(* CoDeSys 2.3 export: DPC_TM10_para.exp *)

(* Data type in Enums *)
TYPE para_e:
(*********************************************)
(*  DON'T MAKE ANY CHANGES TO THIS ENUMS!!   *)
(*    FILE WAS AUTOMATICALLY GENERATED!!     *)
(*********************************************)
(
(* Basic *)
   EEP_number_1_1_1_e          := 790,      (* 0  (0 - 2) *)
   EEP_Input_to_Output_Mode_e  := 770,      (* Not Active  (0 - 2) *)
   EEP_test_par_new_e          := 773,      (* Not Active  (0 - 2) *)
   EEP_test_params_e           := 771,      (* Not Active  (0 - 2) *)
   EEP_test_par2_e             := 772,      (* Not Active  (0 - 2) *)

(* Test Type *)
   EEP_Trimming_type_e         := 818,      (* 53  (0 - 511) *)
   EEP_Analog_type_e           := 819,      (* 245  (53 - ) *)
   EEP_Curve_Type_e            := 820,      (* 245  (66 - 67) *)
   EEP_Function_Type_e         := 821,      (* 248  (248 - 254) *)
   EEP_Percent_Type_e          := 822,      (* 0 % (0 - 1000) *)
   EEP_Ramp_Type_e             := 823,      (* 0 % (0 - 100) *)
   EEP_Switch_Type_e           := 824,      (* 1  ( - ) *)
   EEP_List_Type_e             := 825,      (* AOC  (3 - 2) *)

(* Test Number *)
   EEP_number_1_3_1_e          := 782,      (* 0 ms (0 - 30000) *)
   EEP_number_1_3_2_e          := 783,      (* 0 ms (0 - 30000) *)
   EEP_number_1_3_3_e          := 784,      (* 0 ms (0 - 30000) *)
   EEP_number_1_3_4_e          := 785,      (* 0 ms (0 - 30000) *)
   EEP_number_1_3_5_e          := 786,      (* 0 ms (0 - 30000) *)
   EEP_number_1_3_6_e          := 787,      (* 0 ms (0 - 30000) *)
   EEP_number_1_3_7_e          := 788,      (* 0 ms (0 - 30000) *)
   EEP_number_1_3_8_e          := 789,      (* 0 ms (0 - 30000) *)

(* Output Cfg 1-8 *)
   EEP_Out_Cfg_01_e            := 832,      (* PWM  (1 - 2) *)
   EEP_Out_Cfg_02_e            := 833,      (* PWM  (1 - 2) *)
   EEP_Out_Cfg_03_e            := 834,      (* PWM  (1 - 2) *)
   EEP_Out_Cfg_04_e            := 835,      (* PWM  (1 - 2) *)
   EEP_Out_Cfg_05_e            := 836,      (* PWM  (1 - 2) *)
   EEP_Out_Cfg_06_e            := 837,      (* PWM  (1 - 2) *)
   EEP_Out_Cfg_07_e            := 838,      (* PWM  (1 - 2) *)
   EEP_Out_Cfg_08_e            := 839,      (* PWM  (1 - 2) *)

(* Output Cfg 9-16 *)
   EEP_Out_Cfg_09_e            := 840,      (* PWM  (1 - 2) *)
   EEP_Out_Cfg_10_e            := 841,      (* PWM  (1 - 2) *)
   EEP_Out_Cfg_11_e            := 842,      (* PWM  (1 - 2) *)
   EEP_Out_Cfg_12_e            := 843,      (* PWM  (1 - 2) *)
   EEP_Out_Cfg_13_e            := 844,      (* PWM  (1 - 2) *)
   EEP_Out_Cfg_14_e            := 845,      (* PWM  (1 - 2) *)
   EEP_Out_Cfg_15_e            := 846,      (* PWM  (1 - 2) *)
   EEP_Out_Cfg_16_e            := 847,      (* PWM  (1 - 2) *)

(* Output Cfg 17-24 *)
   EEP_Out_Cfg_17_e            := 848,      (* PWM  (1 - 2) *)
   EEP_Out_Cfg_18_e            := 849,      (* PWM  (1 - 2) *)
   EEP_Out_Cfg_19_e            := 850,      (* Not Active  (0 - 2) *)
   EEP_Out_Cfg_20_e            := 851,      (* Not Active  (0 - 2) *)
   EEP_Out_Cfg_21_e            := 852,      (* Not Active  (0 - 2) *)
   EEP_Out_Cfg_22_e            := 853,      (* Not Active  (0 - 2) *)
   EEP_Out_Cfg_23_e            := 854,      (* Not Active  (0 - 2) *)
   EEP_Out_Cfg_24_e            := 855,      (* Not Active  (0 - 2) *)

(* Output Cfg 25-32 *)
   EEP_Out_Cfg_25_e            := 856,      (* Not Active  (0 - 2) *)
   EEP_Out_Cfg_26_e            := 857,      (* Not Active  (0 - 2) *)
   EEP_Out_Cfg_27_e            := 858,      (* Not Active  (0 - 2) *)
   EEP_Out_Cfg_28_e            := 859,      (* Not Active  (0 - 2) *)
   EEP_Out_Cfg_29_e            := 860,      (* Not Active  (0 - 2) *)
   EEP_Out_Cfg_30_e            := 861,      (* Not Active  (0 - 2) *)
   EEP_Out_Cfg_31_e            := 862,      (* Not Active  (0 - 2) *)
   EEP_Out_Cfg_32_e            := 863,      (* Not Active  (0 - 2) *)

(* Output Cfg 33-40 *)
   EEP_Out_Cfg_33_e            := 864,      (* PWM  (2 - 2) *)
   EEP_Out_Cfg_34_e            := 865,      (* PWM  (2 - 2) *)
   EEP_Out_Cfg_35_e            := 866,      (* PWM  (2 - 2) *)
   EEP_Out_Cfg_36_e            := 867,      (* PWM  (2 - 2) *)
   EEP_Out_Cfg_37_e            := 868,      (* PWM  (1 - 2) *)
   EEP_Out_Cfg_38_e            := 869,      (* PWM  (1 - 2) *)
   EEP_Out_Cfg_39_e            := 870,      (* PWM  (1 - 2) *)
   EEP_Out_Cfg_40_e            := 871,      (* PWM  (1 - 2) *)

(* Output Cfg 41-47 *)
   EEP_Out_Cfg_41_e            := 872,      (* PWM  (1 - 2) *)
   EEP_Out_Cfg_42_e            := 873,      (* PWM  (1 - 2) *)
   EEP_Out_Cfg_43_e            := 874,      (* PWM  (1 - 2) *)
   EEP_Out_Cfg_44_e            := 875,      (* PWM  (1 - 2) *)
   EEP_Out_Cfg_45_e            := 876,      (* PWM  (1 - 2) *)
   EEP_Out_Cfg_46_e            := 877,      (* PWM  (1 - 2) *)
   EEP_Out_Cfg_47_e            := 878,      (* AOV  (3 - 2) *)

(* AOV Configuration *)
   EEP_AOV_Debounce_e          := 880,      (* 200 ms (50 - 250) *)
   EEP_AOV_Freq_e              := 881,      (* 80  (0 - 5000) *)
   EEP_AOV_Res_Min_e           := 882,      (* 0 Ohm (0 - 3000) *)
   EEP_AOV_Res_Max_e           := 883,      (* 0 Ohm (0 - 3000) *)
   EEP_AOV_Kp_e                := 884,      (* 250  (0 - 2000) *)
   EEP_AOV_Ki_e                := 885,      (* 250  (0 - 500) *)

(* AOC Configuration *)
   EEP_AOC_Debounce_e          := 888,      (* 200 ms (50 - 250) *)
   EEP_AOC_Freq_e              := 889,      (* 5000  (0 - 5000) *)
   EEP_AOC_Res_Min_e           := 890,      (* 0 Ohm (0 - 3000) *)
   EEP_AOC_Res_Max_e           := 891,      (* 0 Ohm (0 - 3000) *)
   EEP_AOC_Kp_e                := 892,      (* 250  (0 - 2000) *)
   EEP_AOC_Ki_e                := 893,      (* 250  (0 - 500) *)

(* Output Value 1-8 *)
   EEP_Out_Val_01_e            := 896,      (* 0 % / mA (0 - 10000) *)
   EEP_Out_Val_02_e            := 897,      (* 0 % / mA (0 - 10000) *)
   EEP_Out_Val_03_e            := 898,      (* 0 % / mA (0 - 10000) *)
   EEP_Out_Val_04_e            := 899,      (* 0 % / mA (0 - 10000) *)
   EEP_Out_Val_05_e            := 900,      (* 0 % / mA (0 - 10000) *)
   EEP_Out_Val_06_e            := 901,      (* 0 % / mA (0 - 10000) *)
   EEP_Out_Val_07_e            := 902,      (* 0 % / mA (0 - 10000) *)
   EEP_Out_Val_08_e            := 903,      (* 0 % / mA (0 - 10000) *)

(* Output Value 9-16 *)
   EEP_Out_Val_09_e            := 904,      (* 0 % / mA (0 - 10000) *)
   EEP_Out_Val_10_e            := 905,      (* 0 % / mA (0 - 10000) *)
   EEP_Out_Val_11_e            := 906,      (* 0 % / mA (0 - 10000) *)
   EEP_Out_Val_12_e            := 907,      (* 0 % / mA (0 - 10000) *)
   EEP_Out_Val_13_e            := 908,      (* 0 % / mA (0 - 10000) *)
   EEP_Out_Val_14_e            := 909,      (* 0 % / mA (0 - 10000) *)
   EEP_Out_Val_15_e            := 910,      (* 0 % / mA (0 - 10000) *)
   EEP_Out_Val_16_e            := 911,      (* 0 % / mA (0 - 10000) *)

(* Output Value 17-36 *)
   EEP_Out_Val_17_e            := 912,      (* 0 % / mA (0 - 10000) *)
   EEP_Out_Val_18_e            := 913,      (* 0 % / mA (0 - 10000) *)
   EEP_Out_Val_33_e            := 916,      (* 0 % / mA (0 - 10000) *)
   EEP_Out_Val_34_e            := 917,      (* 0 % / mA (0 - 10000) *)
   EEP_Out_Val_35_e            := 918,      (* 0 % / mA (0 - 10000) *)
   EEP_Out_Val_36_e            := 919,      (* 0 % / mA (0 - 10000) *)

(* Output Value 37-44 *)
   EEP_Out_Val_37_e            := 920,      (* 0 % / mA (0 - 10000) *)
   EEP_Out_Val_38_e            := 921,      (* 0 % / mA (0 - 10000) *)
   EEP_Out_Val_39_e            := 922,      (* 0 % / mA (0 - 10000) *)
   EEP_Out_Val_40_e            := 923,      (* 0 % / mA (0 - 10000) *)
   EEP_Out_Val_41_e            := 924,      (* 0 % / mA (0 - 10000) *)
   EEP_Out_Val_42_e            := 925,      (* 0 % / mA (0 - 10000) *)
   EEP_Out_Val_43_e            := 926,      (* 0 % / mA (0 - 10000) *)
   EEP_Out_Val_44_e            := 927,      (* 0 % / mA (0 - 10000) *)

(* Output Value 45-47 *)
   EEP_Out_Val_45_e            := 928,      (* 0 % / mA (0 - 10000) *)
   EEP_Out_Val_46_e            := 929,      (* 0 % / mA (0 - 10000) *)
   EEP_Out_Val_47_e            := 930,      (* 0 % / mA (0 - 20000) *)

(* POH Configuration *)
   EEP_POH_Debounce_e          := 936,      (* 100 ms (50 - 250) *)
   EEP_POH_Res_Min_e           := 938,      (* 2 Ohm (0 - 3000) *)
   EEP_POH_Res_Max_e           := 939,      (* 52 Ohm (0 - 3000) *)
   EEP_POH_Kp_e                := 940,      (* 250  (0 - 2000) *)
   EEP_POH_Ki_e                := 941,      (* 250  (0 - 500) *)

(* POL Configuration *)
   EEP_POL_Debounce_e          := 944,      (* 100 ms (50 - 250) *)
   EEP_POL_Res_Min_e           := 946,      (* 2 Ohm (0 - 3000) *)
   EEP_POL_Res_Max_e           := 947,      (* 52 Ohm (0 - 3000) *)
   EEP_POL_Kp_e                := 948,      (* 250  (0 - 2000) *)
   EEP_POL_Ki_e                := 949,      (* 250  (0 - 500) *)

(* DOH Configuration *)
   EEP_DOH_Debounce_e          := 952,      (* 200 ms (50 - 250) *)
   EEP_DOH_Res_Min_e           := 954,      (* 6 Ohm (0 - 3000) *)
   EEP_DOH_Res_Max_e           := 955       (* 44 Ohm (0 - 3000) *)

);
END_TYPE

(* Data type in Structures *)
TYPE para_ts:
(***********************************************)
(*  DON'T MAKE ANY CHANGES TO THIS STRUCTURE!! *)
(*      FILE WAS AUTOMATICALLY GENERATED!!     *)
(***********************************************)
STRUCT

(* Basic *)
   number_1_1_1_s16        : INT;           (* 0  (0 - 2) *)
   Input_to_Output_Mode_s16: INT;           (* Not Active  (0 - 2) *)
   test_par_new_s16        : INT;           (* Not Active  (0 - 2) *)
   test_params_s16         : INT;           (* Not Active  (0 - 2) *)
   test_par2_s16           : INT;           (* Not Active  (0 - 2) *)

(* Test Type *)
   Trimming_type_s16       : INT;           (* 53  (0 - 511) *)
   Analog_type_s16         : INT;           (* 245  (53 - ) *)
   Curve_Type_s16          : INT;           (* 245  (66 - 67) *)
   Function_Type_s16       : INT;           (* 248  (248 - 254) *)
   Percent_Type_s16        : INT;           (* 0 % (0 - 1000) *)
   Ramp_Type_s16           : INT;           (* 0 % (0 - 100) *)
   Switch_Type_s16         : INT;           (* 1  ( - ) *)
   List_Type_s16           : INT;           (* AOC  (3 - 2) *)

(* Test Number *)
   number_1_3_1_s16        : INT;           (* 0 ms (0 - 30000) *)
   number_1_3_2_s16        : INT;           (* 0 ms (0 - 30000) *)
   number_1_3_3_s16        : INT;           (* 0 ms (0 - 30000) *)
   number_1_3_4_s16        : INT;           (* 0 ms (0 - 30000) *)
   number_1_3_5_s16        : INT;           (* 0 ms (0 - 30000) *)
   number_1_3_6_s16        : INT;           (* 0 ms (0 - 30000) *)
   number_1_3_7_s16        : INT;           (* 0 ms (0 - 30000) *)
   number_1_3_8_s16        : INT;           (* 0 ms (0 - 30000) *)

(* Output Cfg 1-8 *)
   Out_Cfg_01_s16          : INT;           (* PWM  (1 - 2) *)
   Out_Cfg_02_s16          : INT;           (* PWM  (1 - 2) *)
   Out_Cfg_03_s16          : INT;           (* PWM  (1 - 2) *)
   Out_Cfg_04_s16          : INT;           (* PWM  (1 - 2) *)
   Out_Cfg_05_s16          : INT;           (* PWM  (1 - 2) *)
   Out_Cfg_06_s16          : INT;           (* PWM  (1 - 2) *)
   Out_Cfg_07_s16          : INT;           (* PWM  (1 - 2) *)
   Out_Cfg_08_s16          : INT;           (* PWM  (1 - 2) *)

(* Output Cfg 9-16 *)
   Out_Cfg_09_s16          : INT;           (* PWM  (1 - 2) *)
   Out_Cfg_10_s16          : INT;           (* PWM  (1 - 2) *)
   Out_Cfg_11_s16          : INT;           (* PWM  (1 - 2) *)
   Out_Cfg_12_s16          : INT;           (* PWM  (1 - 2) *)
   Out_Cfg_13_s16          : INT;           (* PWM  (1 - 2) *)
   Out_Cfg_14_s16          : INT;           (* PWM  (1 - 2) *)
   Out_Cfg_15_s16          : INT;           (* PWM  (1 - 2) *)
   Out_Cfg_16_s16          : INT;           (* PWM  (1 - 2) *)

(* Output Cfg 17-24 *)
   Out_Cfg_17_s16          : INT;           (* PWM  (1 - 2) *)
   Out_Cfg_18_s16          : INT;           (* PWM  (1 - 2) *)
   Out_Cfg_19_s16          : INT;           (* Not Active  (0 - 2) *)
   Out_Cfg_20_s16          : INT;           (* Not Active  (0 - 2) *)
   Out_Cfg_21_s16          : INT;           (* Not Active  (0 - 2) *)
   Out_Cfg_22_s16          : INT;           (* Not Active  (0 - 2) *)
   Out_Cfg_23_s16          : INT;           (* Not Active  (0 - 2) *)
   Out_Cfg_24_s16          : INT;           (* Not Active  (0 - 2) *)

(* Output Cfg 25-32 *)
   Out_Cfg_25_s16          : INT;           (* Not Active  (0 - 2) *)
   Out_Cfg_26_s16          : INT;           (* Not Active  (0 - 2) *)
   Out_Cfg_27_s16          : INT;           (* Not Active  (0 - 2) *)
   Out_Cfg_28_s16          : INT;           (* Not Active  (0 - 2) *)
   Out_Cfg_29_s16          : INT;           (* Not Active  (0 - 2) *)
   Out_Cfg_30_s16          : INT;           (* Not Active  (0 - 2) *)
   Out_Cfg_31_s16          : INT;           (* Not Active  (0 - 2) *)
   Out_Cfg_32_s16          : INT;           (* Not Active  (0 - 2) *)

(* Output Cfg 33-40 *)
   Out_Cfg_33_s16          : INT;           (* PWM  (2 - 2) *)
   Out_Cfg_34_s16          : INT;           (* PWM  (2 - 2) *)
   Out_Cfg_35_s16          : INT;           (* PWM  (2 - 2) *)
   Out_Cfg_36_s16          : INT;           (* PWM  (2 - 2) *)
   Out_Cfg_37_s16          : INT;           (* PWM  (1 - 2) *)
   Out_Cfg_38_s16          : INT;           (* PWM  (1 - 2) *)
   Out_Cfg_39_s16          : INT;           (* PWM  (1 - 2) *)
   Out_Cfg_40_s16          : INT;           (* PWM  (1 - 2) *)

(* Output Cfg 41-47 *)
   Out_Cfg_41_s16          : INT;           (* PWM  (1 - 2) *)
   Out_Cfg_42_s16          : INT;           (* PWM  (1 - 2) *)
   Out_Cfg_43_s16          : INT;           (* PWM  (1 - 2) *)
   Out_Cfg_44_s16          : INT;           (* PWM  (1 - 2) *)
   Out_Cfg_45_s16          : INT;           (* PWM  (1 - 2) *)
   Out_Cfg_46_s16          : INT;           (* PWM  (1 - 2) *)
   Out_Cfg_47_s16          : INT;           (* AOV  (3 - 2) *)

(* AOV Configuration *)
   AOV_Debounce_s16        : INT;           (* 200 ms (50 - 250) *)
   AOV_Freq_s16            : INT;           (* 80  (0 - 5000) *)
   AOV_Res_Min_s16         : INT;           (* 0 Ohm (0 - 3000) *)
   AOV_Res_Max_s16         : INT;           (* 0 Ohm (0 - 3000) *)
   AOV_Kp_s16              : INT;           (* 250  (0 - 2000) *)
   AOV_Ki_s16              : INT;           (* 250  (0 - 500) *)

(* AOC Configuration *)
   AOC_Debounce_s16        : INT;           (* 200 ms (50 - 250) *)
   AOC_Freq_s16            : INT;           (* 5000  (0 - 5000) *)
   AOC_Res_Min_s16         : INT;           (* 0 Ohm (0 - 3000) *)
   AOC_Res_Max_s16         : INT;           (* 0 Ohm (0 - 3000) *)
   AOC_Kp_s16              : INT;           (* 250  (0 - 2000) *)
   AOC_Ki_s16              : INT;           (* 250  (0 - 500) *)

(* Output Value 1-8 *)
   Out_Val_01_s16          : INT;           (* 0 % / mA (0 - 10000) *)
   Out_Val_02_s16          : INT;           (* 0 % / mA (0 - 10000) *)
   Out_Val_03_s16          : INT;           (* 0 % / mA (0 - 10000) *)
   Out_Val_04_s16          : INT;           (* 0 % / mA (0 - 10000) *)
   Out_Val_05_s16          : INT;           (* 0 % / mA (0 - 10000) *)
   Out_Val_06_s16          : INT;           (* 0 % / mA (0 - 10000) *)
   Out_Val_07_s16          : INT;           (* 0 % / mA (0 - 10000) *)
   Out_Val_08_s16          : INT;           (* 0 % / mA (0 - 10000) *)

(* Output Value 9-16 *)
   Out_Val_09_s16          : INT;           (* 0 % / mA (0 - 10000) *)
   Out_Val_10_s16          : INT;           (* 0 % / mA (0 - 10000) *)
   Out_Val_11_s16          : INT;           (* 0 % / mA (0 - 10000) *)
   Out_Val_12_s16          : INT;           (* 0 % / mA (0 - 10000) *)
   Out_Val_13_s16          : INT;           (* 0 % / mA (0 - 10000) *)
   Out_Val_14_s16          : INT;           (* 0 % / mA (0 - 10000) *)
   Out_Val_15_s16          : INT;           (* 0 % / mA (0 - 10000) *)
   Out_Val_16_s16          : INT;           (* 0 % / mA (0 - 10000) *)

(* Output Value 17-36 *)
   Out_Val_17_s16          : INT;           (* 0 % / mA (0 - 10000) *)
   Out_Val_18_s16          : INT;           (* 0 % / mA (0 - 10000) *)
   Out_Val_33_s16          : INT;           (* 0 % / mA (0 - 10000) *)
   Out_Val_34_s16          : INT;           (* 0 % / mA (0 - 10000) *)
   Out_Val_35_s16          : INT;           (* 0 % / mA (0 - 10000) *)
   Out_Val_36_s16          : INT;           (* 0 % / mA (0 - 10000) *)

(* Output Value 37-44 *)
   Out_Val_37_s16          : INT;           (* 0 % / mA (0 - 10000) *)
   Out_Val_38_s16          : INT;           (* 0 % / mA (0 - 10000) *)
   Out_Val_39_s16          : INT;           (* 0 % / mA (0 - 10000) *)
   Out_Val_40_s16          : INT;           (* 0 % / mA (0 - 10000) *)
   Out_Val_41_s16          : INT;           (* 0 % / mA (0 - 10000) *)
   Out_Val_42_s16          : INT;           (* 0 % / mA (0 - 10000) *)
   Out_Val_43_s16          : INT;           (* 0 % / mA (0 - 10000) *)
   Out_Val_44_s16          : INT;           (* 0 % / mA (0 - 10000) *)

(* Output Value 45-47 *)
   Out_Val_45_s16          : INT;           (* 0 % / mA (0 - 10000) *)
   Out_Val_46_s16          : INT;           (* 0 % / mA (0 - 10000) *)
   Out_Val_47_s16          : INT;           (* 0 % / mA (0 - 20000) *)

(* POH Configuration *)
   POH_Debounce_s16        : INT;           (* 100 ms (50 - 250) *)
   POH_Res_Min_s16         : INT;           (* 2 Ohm (0 - 3000) *)
   POH_Res_Max_s16         : INT;           (* 52 Ohm (0 - 3000) *)
   POH_Kp_s16              : INT;           (* 250  (0 - 2000) *)
   POH_Ki_s16              : INT;           (* 250  (0 - 500) *)

(* POL Configuration *)
   POL_Debounce_s16        : INT;           (* 100 ms (50 - 250) *)
   POL_Res_Min_s16         : INT;           (* 2 Ohm (0 - 3000) *)
   POL_Res_Max_s16         : INT;           (* 52 Ohm (0 - 3000) *)
   POL_Kp_s16              : INT;           (* 250  (0 - 2000) *)
   POL_Ki_s16              : INT;           (* 250  (0 - 500) *)

(* DOH Configuration *)
   DOH_Debounce_s16        : INT;           (* 200 ms (50 - 250) *)
   DOH_Res_Min_s16         : INT;           (* 6 Ohm (0 - 3000) *)
   DOH_Res_Max_s16         : INT;           (* 44 Ohm (0 - 3000) *)
END_STRUCT
END_TYPE

(* POU Autocode/Callback_diag_getPara, ST *)
PROGRAM Callback_diag_getPara
VAR
   eep:  ARRAY [0..1280] OF INT;
END_VAR
(*********************************************)
(*  DON'T MAKE ANY CHANGES TO THIS PROGRAM!! *)
(*     FILE WAS AUTOMATICALLY GENERATED!!    *)
(*********************************************)

(* get EEPROM pages 0..4 *)
ree_getArray( PAGE0, 0, ADR(eep[0]),    256 );
ree_getArray( PAGE1, 0, ADR(eep[256]),  256 );
ree_getArray( PAGE2, 0, ADR(eep[512]),  256 );
ree_getArray( PAGE3, 0, ADR(eep[768]),  256 );
ree_getArray( PAGE4, 0, ADR(eep[1024]), 256 );

(* Basic *)
para_s.number_1_1_1_s16         := eep[EEP_number_1_1_1_e];
para_s.Input_to_Output_Mode_s16 := eep[EEP_Input_to_Output_Mode_e];
para_s.test_par_new_s16         := eep[EEP_test_par_new_e];
para_s.test_params_s16          := eep[EEP_test_params_e];
para_s.test_par2_s16            := eep[EEP_test_par2_e];

(* Test Type *)
para_s.Trimming_type_s16        := eep[EEP_Trimming_type_e];
para_s.Analog_type_s16          := eep[EEP_Analog_type_e];
para_s.Curve_Type_s16           := eep[EEP_Curve_Type_e];
para_s.Function_Type_s16        := eep[EEP_Function_Type_e];
para_s.Percent_Type_s16         := eep[EEP_Percent_Type_e];
para_s.Ramp_Type_s16            := eep[EEP_Ramp_Type_e];
para_s.Switch_Type_s16          := eep[EEP_Switch_Type_e];
para_s.List_Type_s16            := eep[EEP_List_Type_e];

(* Test Number *)
para_s.number_1_3_1_s16         := eep[EEP_number_1_3_1_e];
para_s.number_1_3_2_s16         := eep[EEP_number_1_3_2_e];
para_s.number_1_3_3_s16         := eep[EEP_number_1_3_3_e];
para_s.number_1_3_4_s16         := eep[EEP_number_1_3_4_e];
para_s.number_1_3_5_s16         := eep[EEP_number_1_3_5_e];
para_s.number_1_3_6_s16         := eep[EEP_number_1_3_6_e];
para_s.number_1_3_7_s16         := eep[EEP_number_1_3_7_e];
para_s.number_1_3_8_s16         := eep[EEP_number_1_3_8_e];

(* Output Cfg 1-8 *)
para_s.Out_Cfg_01_s16           := eep[EEP_Out_Cfg_01_e];
para_s.Out_Cfg_02_s16           := eep[EEP_Out_Cfg_02_e];
para_s.Out_Cfg_03_s16           := eep[EEP_Out_Cfg_03_e];
para_s.Out_Cfg_04_s16           := eep[EEP_Out_Cfg_04_e];
para_s.Out_Cfg_05_s16           := eep[EEP_Out_Cfg_05_e];
para_s.Out_Cfg_06_s16           := eep[EEP_Out_Cfg_06_e];
para_s.Out_Cfg_07_s16           := eep[EEP_Out_Cfg_07_e];
para_s.Out_Cfg_08_s16           := eep[EEP_Out_Cfg_08_e];

(* Output Cfg 9-16 *)
para_s.Out_Cfg_09_s16           := eep[EEP_Out_Cfg_09_e];
para_s.Out_Cfg_10_s16           := eep[EEP_Out_Cfg_10_e];
para_s.Out_Cfg_11_s16           := eep[EEP_Out_Cfg_11_e];
para_s.Out_Cfg_12_s16           := eep[EEP_Out_Cfg_12_e];
para_s.Out_Cfg_13_s16           := eep[EEP_Out_Cfg_13_e];
para_s.Out_Cfg_14_s16           := eep[EEP_Out_Cfg_14_e];
para_s.Out_Cfg_15_s16           := eep[EEP_Out_Cfg_15_e];
para_s.Out_Cfg_16_s16           := eep[EEP_Out_Cfg_16_e];

(* Output Cfg 17-24 *)
para_s.Out_Cfg_17_s16           := eep[EEP_Out_Cfg_17_e];
para_s.Out_Cfg_18_s16           := eep[EEP_Out_Cfg_18_e];
para_s.Out_Cfg_19_s16           := eep[EEP_Out_Cfg_19_e];
para_s.Out_Cfg_20_s16           := eep[EEP_Out_Cfg_20_e];
para_s.Out_Cfg_21_s16           := eep[EEP_Out_Cfg_21_e];
para_s.Out_Cfg_22_s16           := eep[EEP_Out_Cfg_22_e];
para_s.Out_Cfg_23_s16           := eep[EEP_Out_Cfg_23_e];
para_s.Out_Cfg_24_s16           := eep[EEP_Out_Cfg_24_e];

(* Output Cfg 25-32 *)
para_s.Out_Cfg_25_s16           := eep[EEP_Out_Cfg_25_e];
para_s.Out_Cfg_26_s16           := eep[EEP_Out_Cfg_26_e];
para_s.Out_Cfg_27_s16           := eep[EEP_Out_Cfg_27_e];
para_s.Out_Cfg_28_s16           := eep[EEP_Out_Cfg_28_e];
para_s.Out_Cfg_29_s16           := eep[EEP_Out_Cfg_29_e];
para_s.Out_Cfg_30_s16           := eep[EEP_Out_Cfg_30_e];
para_s.Out_Cfg_31_s16           := eep[EEP_Out_Cfg_31_e];
para_s.Out_Cfg_32_s16           := eep[EEP_Out_Cfg_32_e];

(* Output Cfg 33-40 *)
para_s.Out_Cfg_33_s16           := eep[EEP_Out_Cfg_33_e];
para_s.Out_Cfg_34_s16           := eep[EEP_Out_Cfg_34_e];
para_s.Out_Cfg_35_s16           := eep[EEP_Out_Cfg_35_e];
para_s.Out_Cfg_36_s16           := eep[EEP_Out_Cfg_36_e];
para_s.Out_Cfg_37_s16           := eep[EEP_Out_Cfg_37_e];
para_s.Out_Cfg_38_s16           := eep[EEP_Out_Cfg_38_e];
para_s.Out_Cfg_39_s16           := eep[EEP_Out_Cfg_39_e];
para_s.Out_Cfg_40_s16           := eep[EEP_Out_Cfg_40_e];

(* Output Cfg 41-47 *)
para_s.Out_Cfg_41_s16           := eep[EEP_Out_Cfg_41_e];
para_s.Out_Cfg_42_s16           := eep[EEP_Out_Cfg_42_e];
para_s.Out_Cfg_43_s16           := eep[EEP_Out_Cfg_43_e];
para_s.Out_Cfg_44_s16           := eep[EEP_Out_Cfg_44_e];
para_s.Out_Cfg_45_s16           := eep[EEP_Out_Cfg_45_e];
para_s.Out_Cfg_46_s16           := eep[EEP_Out_Cfg_46_e];
para_s.Out_Cfg_47_s16           := eep[EEP_Out_Cfg_47_e];

(* AOV Configuration *)
para_s.AOV_Debounce_s16         := eep[EEP_AOV_Debounce_e];
para_s.AOV_Freq_s16             := eep[EEP_AOV_Freq_e];
para_s.AOV_Res_Min_s16          := eep[EEP_AOV_Res_Min_e];
para_s.AOV_Res_Max_s16          := eep[EEP_AOV_Res_Max_e];
para_s.AOV_Kp_s16               := eep[EEP_AOV_Kp_e];
para_s.AOV_Ki_s16               := eep[EEP_AOV_Ki_e];

(* AOC Configuration *)
para_s.AOC_Debounce_s16         := eep[EEP_AOC_Debounce_e];
para_s.AOC_Freq_s16             := eep[EEP_AOC_Freq_e];
para_s.AOC_Res_Min_s16          := eep[EEP_AOC_Res_Min_e];
para_s.AOC_Res_Max_s16          := eep[EEP_AOC_Res_Max_e];
para_s.AOC_Kp_s16               := eep[EEP_AOC_Kp_e];
para_s.AOC_Ki_s16               := eep[EEP_AOC_Ki_e];

(* Output Value 1-8 *)
para_s.Out_Val_01_s16           := eep[EEP_Out_Val_01_e];
para_s.Out_Val_02_s16           := eep[EEP_Out_Val_02_e];
para_s.Out_Val_03_s16           := eep[EEP_Out_Val_03_e];
para_s.Out_Val_04_s16           := eep[EEP_Out_Val_04_e];
para_s.Out_Val_05_s16           := eep[EEP_Out_Val_05_e];
para_s.Out_Val_06_s16           := eep[EEP_Out_Val_06_e];
para_s.Out_Val_07_s16           := eep[EEP_Out_Val_07_e];
para_s.Out_Val_08_s16           := eep[EEP_Out_Val_08_e];

(* Output Value 9-16 *)
para_s.Out_Val_09_s16           := eep[EEP_Out_Val_09_e];
para_s.Out_Val_10_s16           := eep[EEP_Out_Val_10_e];
para_s.Out_Val_11_s16           := eep[EEP_Out_Val_11_e];
para_s.Out_Val_12_s16           := eep[EEP_Out_Val_12_e];
para_s.Out_Val_13_s16           := eep[EEP_Out_Val_13_e];
para_s.Out_Val_14_s16           := eep[EEP_Out_Val_14_e];
para_s.Out_Val_15_s16           := eep[EEP_Out_Val_15_e];
para_s.Out_Val_16_s16           := eep[EEP_Out_Val_16_e];

(* Output Value 17-36 *)
para_s.Out_Val_17_s16           := eep[EEP_Out_Val_17_e];
para_s.Out_Val_18_s16           := eep[EEP_Out_Val_18_e];
para_s.Out_Val_33_s16           := eep[EEP_Out_Val_33_e];
para_s.Out_Val_34_s16           := eep[EEP_Out_Val_34_e];
para_s.Out_Val_35_s16           := eep[EEP_Out_Val_35_e];
para_s.Out_Val_36_s16           := eep[EEP_Out_Val_36_e];

(* Output Value 37-44 *)
para_s.Out_Val_37_s16           := eep[EEP_Out_Val_37_e];
para_s.Out_Val_38_s16           := eep[EEP_Out_Val_38_e];
para_s.Out_Val_39_s16           := eep[EEP_Out_Val_39_e];
para_s.Out_Val_40_s16           := eep[EEP_Out_Val_40_e];
para_s.Out_Val_41_s16           := eep[EEP_Out_Val_41_e];
para_s.Out_Val_42_s16           := eep[EEP_Out_Val_42_e];
para_s.Out_Val_43_s16           := eep[EEP_Out_Val_43_e];
para_s.Out_Val_44_s16           := eep[EEP_Out_Val_44_e];

(* Output Value 45-47 *)
para_s.Out_Val_45_s16           := eep[EEP_Out_Val_45_e];
para_s.Out_Val_46_s16           := eep[EEP_Out_Val_46_e];
para_s.Out_Val_47_s16           := eep[EEP_Out_Val_47_e];

(* POH Configuration *)
para_s.POH_Debounce_s16         := eep[EEP_POH_Debounce_e];
para_s.POH_Res_Min_s16          := eep[EEP_POH_Res_Min_e];
para_s.POH_Res_Max_s16          := eep[EEP_POH_Res_Max_e];
para_s.POH_Kp_s16               := eep[EEP_POH_Kp_e];
para_s.POH_Ki_s16               := eep[EEP_POH_Ki_e];

(* POL Configuration *)
para_s.POL_Debounce_s16         := eep[EEP_POL_Debounce_e];
para_s.POL_Res_Min_s16          := eep[EEP_POL_Res_Min_e];
para_s.POL_Res_Max_s16          := eep[EEP_POL_Res_Max_e];
para_s.POL_Kp_s16               := eep[EEP_POL_Kp_e];
para_s.POL_Ki_s16               := eep[EEP_POL_Ki_e];

(* DOH Configuration *)
para_s.DOH_Debounce_s16         := eep[EEP_DOH_Debounce_e];
para_s.DOH_Res_Min_s16          := eep[EEP_DOH_Res_Min_e];
para_s.DOH_Res_Max_s16          := eep[EEP_DOH_Res_Max_e];
END_PROGRAM

(* POU Autocode/PrmData, ST *)
PROGRAM PrmData
(*********************************************)
(*  DON'T MAKE ANY CHANGES TO THIS PROGRAM!! *)
(*     FILE WAS AUTOMATICALLY GENERATED!!    *)
(*********************************************)

VAR
END_VAR
VAR CONSTANT

(**)
(*********************************************)
nrPrmMenus_u8          : USINT := 5;

(*********************************************)
(* Parameters Tree *)
(*********************************************)

ParameterMenus_as      : ARRAY [1..5] OF ParameterMenu_ts := 

   (*********************************************)
   (* parameter menu 1 - up to 8 groups can be defined here *)
   (*********************************************)
   (
      MenuName_as8        := 'Menu 1',

      ParameterGroup_as   := 

      (*********************************************)
      (* parameter group 1.1 - up to 8 parameters can be defined here *)
      (*********************************************)
      (
         GroupName_as8   := 'Basic',

         Param_as        := 

         (*********************************************)
         (* parameter 1.1.1 *)
         (*********************************************)
         (
            ParameterName_as8    := 'List test 1',
            ParameterType_u8     := 0,
            attr1_u              := 0,
            attr2_u              := 2,
            UnitCode_au8         := 0,
            AccesslevelCode_u8   := 129,
            attr4_u              := 0,
            EEPROMAddress_s      := (Page_u8 := 3, IntIndex_u8 := 22)
         ),

         (*********************************************)
         (* parameter 1.1.2 *)
         (*********************************************)
         (
            ParameterName_as8    := 'Input_to_Output_Mode',
            ParameterType_u8     := 7,
            attr1_u              := 0,
            attr2_u              := 2,
            UnitCode_au8         := 0,
            AccesslevelCode_u8   := 129,
            attr4_u              := 0,
            EEPROMAddress_s      := (Page_u8 := 3, IntIndex_u8 := 2)
         ),

         (*********************************************)
         (* parameter 1.1.3 *)
         (*********************************************)
         (
         ),

         (*********************************************)
         (* parameter 1.1.4 *)
         (*********************************************)
         (
            ParameterName_as8    := 'Test parameter new',
            ParameterType_u8     := 7,
            attr1_u              := 0,
            attr2_u              := 2,
            UnitCode_au8         := 0,
            AccesslevelCode_u8   := 129,
            attr4_u              := 0,
            EEPROMAddress_s      := (Page_u8 := 3, IntIndex_u8 := 5)
         ),

         (*********************************************)
         (* parameter 1.1.5 *)
         (*********************************************)
         (
         ),

         (*********************************************)
         (* parameter 1.1.6 *)
         (*********************************************)
         (
            ParameterName_as8    := 'Test_parameter',
            ParameterType_u8     := 7,
            attr1_u              := 0,
            attr2_u              := 2,
            UnitCode_au8         := 0,
            AccesslevelCode_u8   := 129,
            attr4_u              := 0,
            EEPROMAddress_s      := (Page_u8 := 3, IntIndex_u8 := 3)
         ),

         (*********************************************)
         (* parameter 1.1.7 *)
         (*********************************************)
         (
         ),

         (*********************************************)
         (* parameter 1.1.8 *)
         (*********************************************)
         (
            ParameterName_as8    := 'Test_params',
            ParameterType_u8     := 7,
            attr1_u              := 0,
            attr2_u              := 2,
            UnitCode_au8         := 0,
            AccesslevelCode_u8   := 129,
            attr4_u              := 0,
            EEPROMAddress_s      := (Page_u8 := 3, IntIndex_u8 := 4)
         )

      ),

      (*********************************************)
      (* parameter group 1.2 - up to 8 parameters can be defined here *)
      (*********************************************)
      (
         GroupName_as8   := 'Test Type',

         Param_as        := 

         (*********************************************)
         (* parameter 1.2.1 *)
         (*********************************************)
         (
            ParameterName_as8    := 'Trimming type',
            ParameterType_u8     := 5,
            attr1_u              := 0,
            attr2_u              := 511,
            UnitCode_au8         := 0,
            AccesslevelCode_u8   := 129,
            attr4_u              := 0,
            EEPROMAddress_s      := (Page_u8 := 3, IntIndex_u8 := 50)
         ),

         (*********************************************)
         (* parameter 1.2.2 *)
         (*********************************************)
         (
            ParameterName_as8    := 'Analog type',
            ParameterType_u8     := 8,
            attr1_u              := 53,
            UnitCode_au8         := 0,
            AccesslevelCode_u8   := 129,
            attr4_u              := 249,
            EEPROMAddress_s      := (Page_u8 := 3, IntIndex_u8 := 51)
         ),

         (*********************************************)
         (* parameter 1.2.3 *)
         (*********************************************)
         (
            ParameterName_as8    := 'Curve Type',
            ParameterType_u8     := 6,
            attr1_u              := 66,
            attr2_u              := 67,
            attr3_u              := 3000,
            UnitCode_au8         := 0,
            AccesslevelCode_u8   := 129,
            attr4_u              := 245,
            EEPROMAddress_s      := (Page_u8 := 3, IntIndex_u8 := 52)
         ),

         (*********************************************)
         (* parameter 1.2.4 *)
         (*********************************************)
         (
            ParameterName_as8    := 'Function Type',
            ParameterType_u8     := 9,
            attr1_u              := 248,
            attr2_u              := 254,
            attr3_u              := 248,
            UnitCode_au8         := 0,
            AccesslevelCode_u8   := 129,
            attr4_u              := 248,
            EEPROMAddress_s      := (Page_u8 := 3, IntIndex_u8 := 53)
         ),

         (*********************************************)
         (* parameter 1.2.5 *)
         (*********************************************)
         (
            ParameterName_as8    := 'Percent Type',
            ParameterType_u8     := 0,
            attr1_u              := 0,
            attr2_u              := 1000,
            attr3_u              := 10,
            UnitCode_au8         := 1,
            Multiplier_s16       := 1,
            Divisor_s16          := 1,
            NumberOfDigits_u16   := 0,
            AccesslevelCode_u8   := 129,
            attr4_u              := 0,
            EEPROMAddress_s      := (Page_u8 := 3, IntIndex_u8 := 54)
         ),

         (*********************************************)
         (* parameter 1.2.6 *)
         (*********************************************)
         (
            ParameterName_as8    := 'Ramp Type',
            ParameterType_u8     := 0,
            attr1_u              := 0,
            attr2_u              := 100,
            attr3_u              := 10,
            UnitCode_au8         := 1,
            Multiplier_s16       := 1,
            Divisor_s16          := 1,
            NumberOfDigits_u16   := 0,
            AccesslevelCode_u8   := 129,
            attr4_u              := 0,
            EEPROMAddress_s      := (Page_u8 := 3, IntIndex_u8 := 55)
         ),

         (*********************************************)
         (* parameter 1.2.7 *)
         (*********************************************)
         (
            ParameterName_as8    := 'Switch Type',
            ParameterType_u8     := 4,
            UnitCode_au8         := 0,
            AccesslevelCode_u8   := 129,
            attr4_u              := 1,
            EEPROMAddress_s      := (Page_u8 := 3, IntIndex_u8 := 56)
         ),

         (*********************************************)
         (* parameter 1.2.8 *)
         (*********************************************)
         (
            ParameterName_as8    := 'List Type',
            ParameterType_u8     := 7,
            attr1_u              := 3,
            attr2_u              := 2,
            UnitCode_au8         := 0,
            AccesslevelCode_u8   := 129,
            attr4_u              := 0,
            EEPROMAddress_s      := (Page_u8 := 3, IntIndex_u8 := 57)
         )

      ),

      (*********************************************)
      (* parameter group 1.3 - up to 8 parameters can be defined here *)
      (*********************************************)
      (
         GroupName_as8   := 'Test Number',

         Param_as        := 

         (*********************************************)
         (* parameter 1.3.1 *)
         (*********************************************)
         (
            ParameterName_as8    := 'Number test 1',
            ParameterType_u8     := 0,
            attr1_u              := 0,
            attr2_u              := 30000,
            attr3_u              := 1,
            UnitCode_au8         := 4,
            Multiplier_s16       := 1,
            Divisor_s16          := 1,
            NumberOfDigits_u16   := 0,
            AccesslevelCode_u8   := 129,
            attr4_u              := 0,
            EEPROMAddress_s      := (Page_u8 := 3, IntIndex_u8 := 14)
         ),

         (*********************************************)
         (* parameter 1.3.2 *)
         (*********************************************)
         (
            ParameterName_as8    := 'Number test 2',
            ParameterType_u8     := 0,
            attr1_u              := 0,
            attr2_u              := 30000,
            attr3_u              := 1,
            UnitCode_au8         := 4,
            Multiplier_s16       := 1,
            Divisor_s16          := 1,
            NumberOfDigits_u16   := 0,
            AccesslevelCode_u8   := 129,
            attr4_u              := 0,
            EEPROMAddress_s      := (Page_u8 := 3, IntIndex_u8 := 15)
         ),

         (*********************************************)
         (* parameter 1.3.3 *)
         (*********************************************)
         (
            ParameterName_as8    := 'Number test 3',
            ParameterType_u8     := 0,
            attr1_u              := 0,
            attr2_u              := 30000,
            attr3_u              := 1,
            UnitCode_au8         := 4,
            Multiplier_s16       := 1,
            Divisor_s16          := 1,
            NumberOfDigits_u16   := 0,
            AccesslevelCode_u8   := 129,
            attr4_u              := 0,
            EEPROMAddress_s      := (Page_u8 := 3, IntIndex_u8 := 16)
         ),

         (*********************************************)
         (* parameter 1.3.4 *)
         (*********************************************)
         (
            ParameterName_as8    := 'Number test 4',
            ParameterType_u8     := 0,
            attr1_u              := 0,
            attr2_u              := 30000,
            attr3_u              := 1,
            UnitCode_au8         := 4,
            Multiplier_s16       := 1,
            Divisor_s16          := 1,
            NumberOfDigits_u16   := 0,
            AccesslevelCode_u8   := 129,
            attr4_u              := 0,
            EEPROMAddress_s      := (Page_u8 := 3, IntIndex_u8 := 17)
         ),

         (*********************************************)
         (* parameter 1.3.5 *)
         (*********************************************)
         (
            ParameterName_as8    := 'Number test 5',
            ParameterType_u8     := 0,
            attr1_u              := 0,
            attr2_u              := 30000,
            attr3_u              := 1,
            UnitCode_au8         := 4,
            Multiplier_s16       := 1,
            Divisor_s16          := 1,
            NumberOfDigits_u16   := 0,
            AccesslevelCode_u8   := 129,
            attr4_u              := 0,
            EEPROMAddress_s      := (Page_u8 := 3, IntIndex_u8 := 18)
         ),

         (*********************************************)
         (* parameter 1.3.6 *)
         (*********************************************)
         (
            ParameterName_as8    := 'Number test 6',
            ParameterType_u8     := 0,
            attr1_u              := 0,
            attr2_u              := 30000,
            attr3_u              := 1,
            UnitCode_au8         := 4,
            Multiplier_s16       := 1,
            Divisor_s16          := 1,
            NumberOfDigits_u16   := 0,
            AccesslevelCode_u8   := 129,
            attr4_u              := 0,
            EEPROMAddress_s      := (Page_u8 := 3, IntIndex_u8 := 19)
         ),

         (*********************************************)
         (* parameter 1.3.7 *)
         (*********************************************)
         (
            ParameterName_as8    := 'Number test 7',
            ParameterType_u8     := 0,
            attr1_u              := 0,
            attr2_u              := 30000,
            attr3_u              := 1,
            UnitCode_au8         := 4,
            Multiplier_s16       := 1,
            Divisor_s16          := 1,
            NumberOfDigits_u16   := 0,
            AccesslevelCode_u8   := 129,
            attr4_u              := 0,
            EEPROMAddress_s      := (Page_u8 := 3, IntIndex_u8 := 20)
         ),

         (*********************************************)
         (* parameter 1.3.8 *)
         (*********************************************)
         (
            ParameterName_as8    := 'Number test 8',
            ParameterType_u8     := 0,
            attr1_u              := 0,
            attr2_u              := 30000,
            attr3_u              := 1,
            UnitCode_au8         := 4,
            Multiplier_s16       := 1,
            Divisor_s16          := 1,
            NumberOfDigits_u16   := 0,
            AccesslevelCode_u8   := 129,
            attr4_u              := 0,
            EEPROMAddress_s      := (Page_u8 := 3, IntIndex_u8 := 21)
         )

      ),

      (*********************************************)
      (* parameter group 1.4 - up to 8 parameters can be defined here *)
      (*********************************************)
      (








      ),

      (*********************************************)
      (* parameter group 1.5 - up to 8 parameters can be defined here *)
      (*********************************************)
      (








      ),

      (*********************************************)
      (* parameter group 1.6 - up to 8 parameters can be defined here *)
      (*********************************************)
      (








      ),

      (*********************************************)
      (* parameter group 1.7 - up to 8 parameters can be defined here *)
      (*********************************************)
      (








      ),

      (*********************************************)
      (* parameter group 1.8 - up to 8 parameters can be defined here *)
      (*********************************************)
      (








      )

   ),

   (*********************************************)
   (* parameter menu 2 - up to 8 groups can be defined here *)
   (*********************************************)
   (
      MenuName_as8        := 'Menu 2',

      ParameterGroup_as   := 

      (*********************************************)
      (* parameter group 2.1 - up to 8 parameters can be defined here *)
      (*********************************************)
      (
         GroupName_as8   := 'Output Cfg 1-8',

         Param_as        := 

         (*********************************************)
         (* parameter 2.1.1 *)
         (*********************************************)
         (
            ParameterName_as8    := 'Output Cfg 1',
            ParameterType_u8     := 7,
            attr1_u              := 1,
            attr2_u              := 2,
            UnitCode_au8         := 0,
            AccesslevelCode_u8   := 129,
            attr4_u              := 0,
            EEPROMAddress_s      := (Page_u8 := 3, IntIndex_u8 := 64)
         ),

         (*********************************************)
         (* parameter 2.1.2 *)
         (*********************************************)
         (
            ParameterName_as8    := 'Output Cfg 2',
            ParameterType_u8     := 7,
            attr1_u              := 1,
            attr2_u              := 2,
            UnitCode_au8         := 0,
            AccesslevelCode_u8   := 129,
            attr4_u              := 0,
            EEPROMAddress_s      := (Page_u8 := 3, IntIndex_u8 := 65)
         ),

         (*********************************************)
         (* parameter 2.1.3 *)
         (*********************************************)
         (
            ParameterName_as8    := 'Output Cfg 3',
            ParameterType_u8     := 7,
            attr1_u              := 1,
            attr2_u              := 2,
            UnitCode_au8         := 0,
            AccesslevelCode_u8   := 129,
            attr4_u              := 0,
            EEPROMAddress_s      := (Page_u8 := 3, IntIndex_u8 := 66)
         ),

         (*********************************************)
         (* parameter 2.1.4 *)
         (*********************************************)
         (
            ParameterName_as8    := 'Output Cfg 4',
            ParameterType_u8     := 7,
            attr1_u              := 1,
            attr2_u              := 2,
            UnitCode_au8         := 0,
            AccesslevelCode_u8   := 129,
            attr4_u              := 0,
            EEPROMAddress_s      := (Page_u8 := 3, IntIndex_u8 := 67)
         ),

         (*********************************************)
         (* parameter 2.1.5 *)
         (*********************************************)
         (
            ParameterName_as8    := 'Output Cfg 5',
            ParameterType_u8     := 7,
            attr1_u              := 1,
            attr2_u              := 2,
            UnitCode_au8         := 0,
            AccesslevelCode_u8   := 129,
            attr4_u              := 0,
            EEPROMAddress_s      := (Page_u8 := 3, IntIndex_u8 := 68)
         ),

         (*********************************************)
         (* parameter 2.1.6 *)
         (*********************************************)
         (
            ParameterName_as8    := 'Output Cfg 6',
            ParameterType_u8     := 7,
            attr1_u              := 1,
            attr2_u              := 2,
            UnitCode_au8         := 0,
            AccesslevelCode_u8   := 129,
            attr4_u              := 0,
            EEPROMAddress_s      := (Page_u8 := 3, IntIndex_u8 := 69)
         ),

         (*********************************************)
         (* parameter 2.1.7 *)
         (*********************************************)
         (
            ParameterName_as8    := 'Output Cfg 7',
            ParameterType_u8     := 7,
            attr1_u              := 1,
            attr2_u              := 2,
            UnitCode_au8         := 0,
            AccesslevelCode_u8   := 129,
            attr4_u              := 0,
            EEPROMAddress_s      := (Page_u8 := 3, IntIndex_u8 := 70)
         ),

         (*********************************************)
         (* parameter 2.1.8 *)
         (*********************************************)
         (
            ParameterName_as8    := 'Output Cfg 8',
            ParameterType_u8     := 7,
            attr1_u              := 1,
            attr2_u              := 2,
            UnitCode_au8         := 0,
            AccesslevelCode_u8   := 129,
            attr4_u              := 0,
            EEPROMAddress_s      := (Page_u8 := 3, IntIndex_u8 := 71)
         )

      ),

      (*********************************************)
      (* parameter group 2.2 - up to 8 parameters can be defined here *)
      (*********************************************)
      (
         GroupName_as8   := 'Output Cfg 9-16',

         Param_as        := 

         (*********************************************)
         (* parameter 2.2.1 *)
         (*********************************************)
         (
            ParameterName_as8    := 'Output Cfg 9',
            ParameterType_u8     := 7,
            attr1_u              := 1,
            attr2_u              := 2,
            UnitCode_au8         := 0,
            AccesslevelCode_u8   := 129,
            attr4_u              := 0,
            EEPROMAddress_s      := (Page_u8 := 3, IntIndex_u8 := 72)
         ),

         (*********************************************)
         (* parameter 2.2.2 *)
         (*********************************************)
         (
            ParameterName_as8    := 'Output Cfg 10',
            ParameterType_u8     := 7,
            attr1_u              := 1,
            attr2_u              := 2,
            UnitCode_au8         := 0,
            AccesslevelCode_u8   := 129,
            attr4_u              := 0,
            EEPROMAddress_s      := (Page_u8 := 3, IntIndex_u8 := 73)
         ),

         (*********************************************)
         (* parameter 2.2.3 *)
         (*********************************************)
         (
            ParameterName_as8    := 'Output Cfg 11',
            ParameterType_u8     := 7,
            attr1_u              := 1,
            attr2_u              := 2,
            UnitCode_au8         := 0,
            AccesslevelCode_u8   := 129,
            attr4_u              := 0,
            EEPROMAddress_s      := (Page_u8 := 3, IntIndex_u8 := 74)
         ),

         (*********************************************)
         (* parameter 2.2.4 *)
         (*********************************************)
         (
            ParameterName_as8    := 'Output Cfg 12',
            ParameterType_u8     := 7,
            attr1_u              := 1,
            attr2_u              := 2,
            UnitCode_au8         := 0,
            AccesslevelCode_u8   := 129,
            attr4_u              := 0,
            EEPROMAddress_s      := (Page_u8 := 3, IntIndex_u8 := 75)
         ),

         (*********************************************)
         (* parameter 2.2.5 *)
         (*********************************************)
         (
            ParameterName_as8    := 'Output Cfg 13',
            ParameterType_u8     := 7,
            attr1_u              := 1,
            attr2_u              := 2,
            UnitCode_au8         := 0,
            AccesslevelCode_u8   := 129,
            attr4_u              := 0,
            EEPROMAddress_s      := (Page_u8 := 3, IntIndex_u8 := 76)
         ),

         (*********************************************)
         (* parameter 2.2.6 *)
         (*********************************************)
         (
            ParameterName_as8    := 'Output Cfg 14',
            ParameterType_u8     := 7,
            attr1_u              := 1,
            attr2_u              := 2,
            UnitCode_au8         := 0,
            AccesslevelCode_u8   := 129,
            attr4_u              := 0,
            EEPROMAddress_s      := (Page_u8 := 3, IntIndex_u8 := 77)
         ),

         (*********************************************)
         (* parameter 2.2.7 *)
         (*********************************************)
         (
            ParameterName_as8    := 'Output Cfg 15',
            ParameterType_u8     := 7,
            attr1_u              := 1,
            attr2_u              := 2,
            UnitCode_au8         := 0,
            AccesslevelCode_u8   := 129,
            attr4_u              := 0,
            EEPROMAddress_s      := (Page_u8 := 3, IntIndex_u8 := 78)
         ),

         (*********************************************)
         (* parameter 2.2.8 *)
         (*********************************************)
         (
            ParameterName_as8    := 'Output Cfg 16',
            ParameterType_u8     := 7,
            attr1_u              := 1,
            attr2_u              := 2,
            UnitCode_au8         := 0,
            AccesslevelCode_u8   := 129,
            attr4_u              := 0,
            EEPROMAddress_s      := (Page_u8 := 3, IntIndex_u8 := 79)
         )

      ),

      (*********************************************)
      (* parameter group 2.3 - up to 8 parameters can be defined here *)
      (*********************************************)
      (
         GroupName_as8   := 'Output Cfg 17-24',

         Param_as        := 

         (*********************************************)
         (* parameter 2.3.1 *)
         (*********************************************)
         (
            ParameterName_as8    := 'Output Cfg 17',
            ParameterType_u8     := 7,
            attr1_u              := 1,
            attr2_u              := 2,
            UnitCode_au8         := 0,
            AccesslevelCode_u8   := 129,
            attr4_u              := 0,
            EEPROMAddress_s      := (Page_u8 := 3, IntIndex_u8 := 80)
         ),

         (*********************************************)
         (* parameter 2.3.2 *)
         (*********************************************)
         (
            ParameterName_as8    := 'Output Cfg 18',
            ParameterType_u8     := 7,
            attr1_u              := 1,
            attr2_u              := 2,
            UnitCode_au8         := 0,
            AccesslevelCode_u8   := 129,
            attr4_u              := 0,
            EEPROMAddress_s      := (Page_u8 := 3, IntIndex_u8 := 81)
         ),

         (*********************************************)
         (* parameter 2.3.3 *)
         (*********************************************)
         (
            ParameterName_as8    := 'Output Cfg 19',
            ParameterType_u8     := 7,
            attr1_u              := 0,
            attr2_u              := 2,
            UnitCode_au8         := 0,
            AccesslevelCode_u8   := 129,
            attr4_u              := 0,
            EEPROMAddress_s      := (Page_u8 := 3, IntIndex_u8 := 82)
         ),

         (*********************************************)
         (* parameter 2.3.4 *)
         (*********************************************)
         (
            ParameterName_as8    := 'Output Cfg 20',
            ParameterType_u8     := 7,
            attr1_u              := 0,
            attr2_u              := 2,
            UnitCode_au8         := 0,
            AccesslevelCode_u8   := 129,
            attr4_u              := 0,
            EEPROMAddress_s      := (Page_u8 := 3, IntIndex_u8 := 83)
         ),

         (*********************************************)
         (* parameter 2.3.5 *)
         (*********************************************)
         (
            ParameterName_as8    := 'Output Cfg 21',
            ParameterType_u8     := 7,
            attr1_u              := 0,
            attr2_u              := 2,
            UnitCode_au8         := 0,
            AccesslevelCode_u8   := 129,
            attr4_u              := 0,
            EEPROMAddress_s      := (Page_u8 := 3, IntIndex_u8 := 84)
         ),

         (*********************************************)
         (* parameter 2.3.6 *)
         (*********************************************)
         (
            ParameterName_as8    := 'Output Cfg 22',
            ParameterType_u8     := 7,
            attr1_u              := 0,
            attr2_u              := 2,
            UnitCode_au8         := 0,
            AccesslevelCode_u8   := 129,
            attr4_u              := 0,
            EEPROMAddress_s      := (Page_u8 := 3, IntIndex_u8 := 85)
         ),

         (*********************************************)
         (* parameter 2.3.7 *)
         (*********************************************)
         (
            ParameterName_as8    := 'Output Cfg 23',
            ParameterType_u8     := 7,
            attr1_u              := 0,
            attr2_u              := 2,
            UnitCode_au8         := 0,
            AccesslevelCode_u8   := 129,
            attr4_u              := 0,
            EEPROMAddress_s      := (Page_u8 := 3, IntIndex_u8 := 86)
         ),

         (*********************************************)
         (* parameter 2.3.8 *)
         (*********************************************)
         (
            ParameterName_as8    := 'Output Cfg 24',
            ParameterType_u8     := 7,
            attr1_u              := 0,
            attr2_u              := 2,
            UnitCode_au8         := 0,
            AccesslevelCode_u8   := 129,
            attr4_u              := 0,
            EEPROMAddress_s      := (Page_u8 := 3, IntIndex_u8 := 87)
         )

      ),

      (*********************************************)
      (* parameter group 2.4 - up to 8 parameters can be defined here *)
      (*********************************************)
      (
         GroupName_as8   := 'Output Cfg 25-32',

         Param_as        := 

         (*********************************************)
         (* parameter 2.4.1 *)
         (*********************************************)
         (
            ParameterName_as8    := 'Output Cfg 25',
            ParameterType_u8     := 7,
            attr1_u              := 0,
            attr2_u              := 2,
            UnitCode_au8         := 0,
            AccesslevelCode_u8   := 129,
            attr4_u              := 0,
            EEPROMAddress_s      := (Page_u8 := 3, IntIndex_u8 := 88)
         ),

         (*********************************************)
         (* parameter 2.4.2 *)
         (*********************************************)
         (
            ParameterName_as8    := 'Output Cfg 26',
            ParameterType_u8     := 7,
            attr1_u              := 0,
            attr2_u              := 2,
            UnitCode_au8         := 0,
            AccesslevelCode_u8   := 129,
            attr4_u              := 0,
            EEPROMAddress_s      := (Page_u8 := 3, IntIndex_u8 := 89)
         ),

         (*********************************************)
         (* parameter 2.4.3 *)
         (*********************************************)
         (
            ParameterName_as8    := 'Output Cfg 27',
            ParameterType_u8     := 7,
            attr1_u              := 0,
            attr2_u              := 2,
            UnitCode_au8         := 0,
            AccesslevelCode_u8   := 129,
            attr4_u              := 0,
            EEPROMAddress_s      := (Page_u8 := 3, IntIndex_u8 := 90)
         ),

         (*********************************************)
         (* parameter 2.4.4 *)
         (*********************************************)
         (
            ParameterName_as8    := 'Output Cfg 28',
            ParameterType_u8     := 7,
            attr1_u              := 0,
            attr2_u              := 2,
            UnitCode_au8         := 0,
            AccesslevelCode_u8   := 129,
            attr4_u              := 0,
            EEPROMAddress_s      := (Page_u8 := 3, IntIndex_u8 := 91)
         ),

         (*********************************************)
         (* parameter 2.4.5 *)
         (*********************************************)
         (
            ParameterName_as8    := 'Output Cfg 29',
            ParameterType_u8     := 7,
            attr1_u              := 0,
            attr2_u              := 2,
            UnitCode_au8         := 0,
            AccesslevelCode_u8   := 129,
            attr4_u              := 0,
            EEPROMAddress_s      := (Page_u8 := 3, IntIndex_u8 := 92)
         ),

         (*********************************************)
         (* parameter 2.4.6 *)
         (*********************************************)
         (
            ParameterName_as8    := 'Output Cfg 30',
            ParameterType_u8     := 7,
            attr1_u              := 0,
            attr2_u              := 2,
            UnitCode_au8         := 0,
            AccesslevelCode_u8   := 129,
            attr4_u              := 0,
            EEPROMAddress_s      := (Page_u8 := 3, IntIndex_u8 := 93)
         ),

         (*********************************************)
         (* parameter 2.4.7 *)
         (*********************************************)
         (
            ParameterName_as8    := 'Output Cfg 31',
            ParameterType_u8     := 7,
            attr1_u              := 0,
            attr2_u              := 2,
            UnitCode_au8         := 0,
            AccesslevelCode_u8   := 129,
            attr4_u              := 0,
            EEPROMAddress_s      := (Page_u8 := 3, IntIndex_u8 := 94)
         ),

         (*********************************************)
         (* parameter 2.4.8 *)
         (*********************************************)
         (
            ParameterName_as8    := 'Output Cfg 32',
            ParameterType_u8     := 7,
            attr1_u              := 0,
            attr2_u              := 2,
            UnitCode_au8         := 0,
            AccesslevelCode_u8   := 129,
            attr4_u              := 0,
            EEPROMAddress_s      := (Page_u8 := 3, IntIndex_u8 := 95)
         )

      ),

      (*********************************************)
      (* parameter group 2.5 - up to 8 parameters can be defined here *)
      (*********************************************)
      (
         GroupName_as8   := 'Output Cfg 33-40',

         Param_as        := 

         (*********************************************)
         (* parameter 2.5.1 *)
         (*********************************************)
         (
            ParameterName_as8    := 'Output Cfg 33',
            ParameterType_u8     := 7,
            attr1_u              := 2,
            attr2_u              := 2,
            UnitCode_au8         := 0,
            AccesslevelCode_u8   := 129,
            attr4_u              := 0,
            EEPROMAddress_s      := (Page_u8 := 3, IntIndex_u8 := 96)
         ),

         (*********************************************)
         (* parameter 2.5.2 *)
         (*********************************************)
         (
            ParameterName_as8    := 'Output Cfg 34',
            ParameterType_u8     := 7,
            attr1_u              := 2,
            attr2_u              := 2,
            UnitCode_au8         := 0,
            AccesslevelCode_u8   := 129,
            attr4_u              := 0,
            EEPROMAddress_s      := (Page_u8 := 3, IntIndex_u8 := 97)
         ),

         (*********************************************)
         (* parameter 2.5.3 *)
         (*********************************************)
         (
            ParameterName_as8    := 'Output Cfg 35',
            ParameterType_u8     := 7,
            attr1_u              := 2,
            attr2_u              := 2,
            UnitCode_au8         := 0,
            AccesslevelCode_u8   := 129,
            attr4_u              := 0,
            EEPROMAddress_s      := (Page_u8 := 3, IntIndex_u8 := 98)
         ),

         (*********************************************)
         (* parameter 2.5.4 *)
         (*********************************************)
         (
            ParameterName_as8    := 'Output Cfg 36',
            ParameterType_u8     := 7,
            attr1_u              := 2,
            attr2_u              := 2,
            UnitCode_au8         := 0,
            AccesslevelCode_u8   := 129,
            attr4_u              := 0,
            EEPROMAddress_s      := (Page_u8 := 3, IntIndex_u8 := 99)
         ),

         (*********************************************)
         (* parameter 2.5.5 *)
         (*********************************************)
         (
            ParameterName_as8    := 'Output Cfg 37',
            ParameterType_u8     := 7,
            attr1_u              := 1,
            attr2_u              := 2,
            UnitCode_au8         := 0,
            AccesslevelCode_u8   := 129,
            attr4_u              := 0,
            EEPROMAddress_s      := (Page_u8 := 3, IntIndex_u8 := 100)
         ),

         (*********************************************)
         (* parameter 2.5.6 *)
         (*********************************************)
         (
            ParameterName_as8    := 'Output Cfg 38',
            ParameterType_u8     := 7,
            attr1_u              := 1,
            attr2_u              := 2,
            UnitCode_au8         := 0,
            AccesslevelCode_u8   := 129,
            attr4_u              := 0,
            EEPROMAddress_s      := (Page_u8 := 3, IntIndex_u8 := 101)
         ),

         (*********************************************)
         (* parameter 2.5.7 *)
         (*********************************************)
         (
            ParameterName_as8    := 'Output Cfg 39',
            ParameterType_u8     := 7,
            attr1_u              := 1,
            attr2_u              := 2,
            UnitCode_au8         := 0,
            AccesslevelCode_u8   := 129,
            attr4_u              := 0,
            EEPROMAddress_s      := (Page_u8 := 3, IntIndex_u8 := 102)
         ),

         (*********************************************)
         (* parameter 2.5.8 *)
         (*********************************************)
         (
            ParameterName_as8    := 'Output Cfg 40',
            ParameterType_u8     := 7,
            attr1_u              := 1,
            attr2_u              := 2,
            UnitCode_au8         := 0,
            AccesslevelCode_u8   := 129,
            attr4_u              := 0,
            EEPROMAddress_s      := (Page_u8 := 3, IntIndex_u8 := 103)
         )

      ),

      (*********************************************)
      (* parameter group 2.6 - up to 8 parameters can be defined here *)
      (*********************************************)
      (
         GroupName_as8   := 'Output Cfg 41-47',

         Param_as        := 

         (*********************************************)
         (* parameter 2.6.1 *)
         (*********************************************)
         (
            ParameterName_as8    := 'Output Cfg 41',
            ParameterType_u8     := 7,
            attr1_u              := 1,
            attr2_u              := 2,
            UnitCode_au8         := 0,
            AccesslevelCode_u8   := 129,
            attr4_u              := 0,
            EEPROMAddress_s      := (Page_u8 := 3, IntIndex_u8 := 104)
         ),

         (*********************************************)
         (* parameter 2.6.2 *)
         (*********************************************)
         (
            ParameterName_as8    := 'Output Cfg 42',
            ParameterType_u8     := 7,
            attr1_u              := 1,
            attr2_u              := 2,
            UnitCode_au8         := 0,
            AccesslevelCode_u8   := 129,
            attr4_u              := 0,
            EEPROMAddress_s      := (Page_u8 := 3, IntIndex_u8 := 105)
         ),

         (*********************************************)
         (* parameter 2.6.3 *)
         (*********************************************)
         (
            ParameterName_as8    := 'Output Cfg 43',
            ParameterType_u8     := 7,
            attr1_u              := 1,
            attr2_u              := 2,
            UnitCode_au8         := 0,
            AccesslevelCode_u8   := 129,
            attr4_u              := 0,
            EEPROMAddress_s      := (Page_u8 := 3, IntIndex_u8 := 106)
         ),

         (*********************************************)
         (* parameter 2.6.4 *)
         (*********************************************)
         (
            ParameterName_as8    := 'Output Cfg 44',
            ParameterType_u8     := 7,
            attr1_u              := 1,
            attr2_u              := 2,
            UnitCode_au8         := 0,
            AccesslevelCode_u8   := 129,
            attr4_u              := 0,
            EEPROMAddress_s      := (Page_u8 := 3, IntIndex_u8 := 107)
         ),

         (*********************************************)
         (* parameter 2.6.5 *)
         (*********************************************)
         (
            ParameterName_as8    := 'Output Cfg 45',
            ParameterType_u8     := 7,
            attr1_u              := 1,
            attr2_u              := 2,
            UnitCode_au8         := 0,
            AccesslevelCode_u8   := 129,
            attr4_u              := 0,
            EEPROMAddress_s      := (Page_u8 := 3, IntIndex_u8 := 108)
         ),

         (*********************************************)
         (* parameter 2.6.6 *)
         (*********************************************)
         (
            ParameterName_as8    := 'Output Cfg 46',
            ParameterType_u8     := 7,
            attr1_u              := 1,
            attr2_u              := 2,
            UnitCode_au8         := 0,
            AccesslevelCode_u8   := 129,
            attr4_u              := 0,
            EEPROMAddress_s      := (Page_u8 := 3, IntIndex_u8 := 109)
         ),

         (*********************************************)
         (* parameter 2.6.7 *)
         (*********************************************)
         (
            ParameterName_as8    := 'Output Cfg 47',
            ParameterType_u8     := 7,
            attr1_u              := 3,
            attr2_u              := 2,
            UnitCode_au8         := 0,
            AccesslevelCode_u8   := 129,
            attr4_u              := 1,
            EEPROMAddress_s      := (Page_u8 := 3, IntIndex_u8 := 110)
         ),

         (*********************************************)
         (* parameter 2.6.8 *)
         (*********************************************)
         (
         )

      ),

      (*********************************************)
      (* parameter group 2.7 - up to 8 parameters can be defined here *)
      (*********************************************)
      (
         GroupName_as8   := 'AOV Configuration',

         Param_as        := 

         (*********************************************)
         (* parameter 2.7.1 *)
         (*********************************************)
         (
            ParameterName_as8    := 'AOV Debounce',
            ParameterType_u8     := 0,
            attr1_u              := 50,
            attr2_u              := 250,
            attr3_u              := 10,
            UnitCode_au8         := 4,
            Multiplier_s16       := 1,
            Divisor_s16          := 1,
            NumberOfDigits_u16   := 0,
            AccesslevelCode_u8   := 179,
            attr4_u              := 200,
            EEPROMAddress_s      := (Page_u8 := 3, IntIndex_u8 := 112)
         ),

         (*********************************************)
         (* parameter 2.7.2 *)
         (*********************************************)
         (
            ParameterName_as8    := 'AOV Frequency',
            ParameterType_u8     := 0,
            attr1_u              := 0,
            attr2_u              := 5000,
            attr3_u              := 10,
            UnitCode_au8         := 0,
            Multiplier_s16       := 1,
            Divisor_s16          := 1,
            NumberOfDigits_u16   := 0,
            AccesslevelCode_u8   := 179,
            attr4_u              := 80,
            EEPROMAddress_s      := (Page_u8 := 3, IntIndex_u8 := 113)
         ),

         (*********************************************)
         (* parameter 2.7.3 *)
         (*********************************************)
         (
            ParameterName_as8    := 'AOV Resistance Min',
            ParameterType_u8     := 0,
            attr1_u              := 0,
            attr2_u              := 3000,
            attr3_u              := 10,
            UnitCode_au8         := 18,
            Multiplier_s16       := 1,
            Divisor_s16          := 1,
            NumberOfDigits_u16   := 0,
            AccesslevelCode_u8   := 179,
            attr4_u              := 0,
            EEPROMAddress_s      := (Page_u8 := 3, IntIndex_u8 := 114)
         ),

         (*********************************************)
         (* parameter 2.7.4 *)
         (*********************************************)
         (
            ParameterName_as8    := 'AOV Resistance Max',
            ParameterType_u8     := 0,
            attr1_u              := 0,
            attr2_u              := 3000,
            attr3_u              := 10,
            UnitCode_au8         := 18,
            Multiplier_s16       := 1,
            Divisor_s16          := 1,
            NumberOfDigits_u16   := 0,
            AccesslevelCode_u8   := 179,
            attr4_u              := 0,
            EEPROMAddress_s      := (Page_u8 := 3, IntIndex_u8 := 115)
         ),

         (*********************************************)
         (* parameter 2.7.5 *)
         (*********************************************)
         (
            ParameterName_as8    := 'AOV Kp',
            ParameterType_u8     := 0,
            attr1_u              := 0,
            attr2_u              := 2000,
            attr3_u              := 50,
            UnitCode_au8         := 0,
            Multiplier_s16       := 1,
            Divisor_s16          := 1,
            NumberOfDigits_u16   := 0,
            AccesslevelCode_u8   := 179,
            attr4_u              := 250,
            EEPROMAddress_s      := (Page_u8 := 3, IntIndex_u8 := 116)
         ),

         (*********************************************)
         (* parameter 2.7.6 *)
         (*********************************************)
         (
            ParameterName_as8    := 'AOV Ki',
            ParameterType_u8     := 0,
            attr1_u              := 0,
            attr2_u              := 500,
            attr3_u              := 50,
            UnitCode_au8         := 0,
            Multiplier_s16       := 1,
            Divisor_s16          := 1,
            NumberOfDigits_u16   := 0,
            AccesslevelCode_u8   := 179,
            attr4_u              := 250,
            EEPROMAddress_s      := (Page_u8 := 3, IntIndex_u8 := 117)
         ),

         (*********************************************)
         (* parameter 2.7.7 *)
         (*********************************************)
         (
         ),

         (*********************************************)
         (* parameter 2.7.8 *)
         (*********************************************)
         (
         )

      ),

      (*********************************************)
      (* parameter group 2.8 - up to 8 parameters can be defined here *)
      (*********************************************)
      (
         GroupName_as8   := 'AOC Configuration',

         Param_as        := 

         (*********************************************)
         (* parameter 2.8.1 *)
         (*********************************************)
         (
            ParameterName_as8    := 'AOC Debounce',
            ParameterType_u8     := 0,
            attr1_u              := 50,
            attr2_u              := 250,
            attr3_u              := 10,
            UnitCode_au8         := 4,
            Multiplier_s16       := 1,
            Divisor_s16          := 1,
            NumberOfDigits_u16   := 0,
            AccesslevelCode_u8   := 179,
            attr4_u              := 200,
            EEPROMAddress_s      := (Page_u8 := 3, IntIndex_u8 := 120)
         ),

         (*********************************************)
         (* parameter 2.8.2 *)
         (*********************************************)
         (
            ParameterName_as8    := 'AOC Frequency',
            ParameterType_u8     := 0,
            attr1_u              := 0,
            attr2_u              := 5000,
            attr3_u              := 10,
            UnitCode_au8         := 0,
            AccesslevelCode_u8   := 179,
            attr4_u              := 5000,
            EEPROMAddress_s      := (Page_u8 := 3, IntIndex_u8 := 121)
         ),

         (*********************************************)
         (* parameter 2.8.3 *)
         (*********************************************)
         (
            ParameterName_as8    := 'AOC Resistance Min',
            ParameterType_u8     := 0,
            attr1_u              := 0,
            attr2_u              := 3000,
            attr3_u              := 10,
            UnitCode_au8         := 18,
            Multiplier_s16       := 1,
            Divisor_s16          := 1,
            NumberOfDigits_u16   := 0,
            AccesslevelCode_u8   := 179,
            attr4_u              := 0,
            EEPROMAddress_s      := (Page_u8 := 3, IntIndex_u8 := 122)
         ),

         (*********************************************)
         (* parameter 2.8.4 *)
         (*********************************************)
         (
            ParameterName_as8    := 'AOC Resistance Max',
            ParameterType_u8     := 0,
            attr1_u              := 0,
            attr2_u              := 3000,
            attr3_u              := 10,
            UnitCode_au8         := 18,
            Multiplier_s16       := 1,
            Divisor_s16          := 1,
            NumberOfDigits_u16   := 0,
            AccesslevelCode_u8   := 179,
            attr4_u              := 0,
            EEPROMAddress_s      := (Page_u8 := 3, IntIndex_u8 := 123)
         ),

         (*********************************************)
         (* parameter 2.8.5 *)
         (*********************************************)
         (
            ParameterName_as8    := 'AOC Kp',
            ParameterType_u8     := 0,
            attr1_u              := 0,
            attr2_u              := 2000,
            attr3_u              := 50,
            UnitCode_au8         := 0,
            Multiplier_s16       := 1,
            Divisor_s16          := 1,
            NumberOfDigits_u16   := 0,
            AccesslevelCode_u8   := 179,
            attr4_u              := 250,
            EEPROMAddress_s      := (Page_u8 := 3, IntIndex_u8 := 124)
         ),

         (*********************************************)
         (* parameter 2.8.6 *)
         (*********************************************)
         (
            ParameterName_as8    := 'AOC Ki',
            ParameterType_u8     := 0,
            attr1_u              := 0,
            attr2_u              := 500,
            attr3_u              := 50,
            UnitCode_au8         := 0,
            Multiplier_s16       := 1,
            Divisor_s16          := 1,
            NumberOfDigits_u16   := 0,
            AccesslevelCode_u8   := 179,
            attr4_u              := 250,
            EEPROMAddress_s      := (Page_u8 := 3, IntIndex_u8 := 125)
         ),

         (*********************************************)
         (* parameter 2.8.7 *)
         (*********************************************)
         (
         ),

         (*********************************************)
         (* parameter 2.8.8 *)
         (*********************************************)
         (
         )

      )

   ),

   (*********************************************)
   (* parameter menu 3 - up to 8 groups can be defined here *)
   (*********************************************)
   (
      MenuName_as8        := 'Menu 3',

      ParameterGroup_as   := 

      (*********************************************)
      (* parameter group 3.1 - up to 8 parameters can be defined here *)
      (*********************************************)
      (
         GroupName_as8   := 'Output Value 1-8',

         Param_as        := 

         (*********************************************)
         (* parameter 3.1.1 *)
         (*********************************************)
         (
            ParameterName_as8    := 'Output Value 1',
            ParameterType_u8     := 0,
            attr1_u              := 0,
            attr2_u              := 10000,
            attr3_u              := 50,
            UnitCode_au8         := 15,
            Multiplier_s16       := 1,
            Divisor_s16          := 1,
            NumberOfDigits_u16   := 0,
            AccesslevelCode_u8   := 129,
            attr4_u              := 0,
            EEPROMAddress_s      := (Page_u8 := 3, IntIndex_u8 := 128)
         ),

         (*********************************************)
         (* parameter 3.1.2 *)
         (*********************************************)
         (
            ParameterName_as8    := 'Output Value 2',
            ParameterType_u8     := 0,
            attr1_u              := 0,
            attr2_u              := 10000,
            attr3_u              := 50,
            UnitCode_au8         := 15,
            Multiplier_s16       := 1,
            Divisor_s16          := 1,
            NumberOfDigits_u16   := 0,
            AccesslevelCode_u8   := 129,
            attr4_u              := 0,
            EEPROMAddress_s      := (Page_u8 := 3, IntIndex_u8 := 129)
         ),

         (*********************************************)
         (* parameter 3.1.3 *)
         (*********************************************)
         (
            ParameterName_as8    := 'Output Value 3',
            ParameterType_u8     := 0,
            attr1_u              := 0,
            attr2_u              := 10000,
            attr3_u              := 50,
            UnitCode_au8         := 15,
            Multiplier_s16       := 1,
            Divisor_s16          := 1,
            NumberOfDigits_u16   := 0,
            AccesslevelCode_u8   := 129,
            attr4_u              := 0,
            EEPROMAddress_s      := (Page_u8 := 3, IntIndex_u8 := 130)
         ),

         (*********************************************)
         (* parameter 3.1.4 *)
         (*********************************************)
         (
            ParameterName_as8    := 'Output Value 4',
            ParameterType_u8     := 0,
            attr1_u              := 0,
            attr2_u              := 10000,
            attr3_u              := 50,
            UnitCode_au8         := 15,
            Multiplier_s16       := 1,
            Divisor_s16          := 1,
            NumberOfDigits_u16   := 0,
            AccesslevelCode_u8   := 129,
            attr4_u              := 0,
            EEPROMAddress_s      := (Page_u8 := 3, IntIndex_u8 := 131)
         ),

         (*********************************************)
         (* parameter 3.1.5 *)
         (*********************************************)
         (
            ParameterName_as8    := 'Output Value 5',
            ParameterType_u8     := 0,
            attr1_u              := 0,
            attr2_u              := 10000,
            attr3_u              := 50,
            UnitCode_au8         := 15,
            Multiplier_s16       := 1,
            Divisor_s16          := 1,
            NumberOfDigits_u16   := 0,
            AccesslevelCode_u8   := 129,
            attr4_u              := 0,
            EEPROMAddress_s      := (Page_u8 := 3, IntIndex_u8 := 132)
         ),

         (*********************************************)
         (* parameter 3.1.6 *)
         (*********************************************)
         (
            ParameterName_as8    := 'Output Value 6',
            ParameterType_u8     := 0,
            attr1_u              := 0,
            attr2_u              := 10000,
            attr3_u              := 50,
            UnitCode_au8         := 15,
            Multiplier_s16       := 1,
            Divisor_s16          := 1,
            NumberOfDigits_u16   := 0,
            AccesslevelCode_u8   := 129,
            attr4_u              := 0,
            EEPROMAddress_s      := (Page_u8 := 3, IntIndex_u8 := 133)
         ),

         (*********************************************)
         (* parameter 3.1.7 *)
         (*********************************************)
         (
            ParameterName_as8    := 'Output Value 7',
            ParameterType_u8     := 0,
            attr1_u              := 0,
            attr2_u              := 10000,
            attr3_u              := 50,
            UnitCode_au8         := 15,
            Multiplier_s16       := 1,
            Divisor_s16          := 1,
            NumberOfDigits_u16   := 0,
            AccesslevelCode_u8   := 129,
            attr4_u              := 0,
            EEPROMAddress_s      := (Page_u8 := 3, IntIndex_u8 := 134)
         ),

         (*********************************************)
         (* parameter 3.1.8 *)
         (*********************************************)
         (
            ParameterName_as8    := 'Output Value 8',
            ParameterType_u8     := 0,
            attr1_u              := 0,
            attr2_u              := 10000,
            attr3_u              := 50,
            UnitCode_au8         := 15,
            Multiplier_s16       := 1,
            Divisor_s16          := 1,
            NumberOfDigits_u16   := 0,
            AccesslevelCode_u8   := 129,
            attr4_u              := 0,
            EEPROMAddress_s      := (Page_u8 := 3, IntIndex_u8 := 135)
         )

      ),

      (*********************************************)
      (* parameter group 3.2 - up to 8 parameters can be defined here *)
      (*********************************************)
      (
         GroupName_as8   := 'Output Value 9-16',

         Param_as        := 

         (*********************************************)
         (* parameter 3.2.1 *)
         (*********************************************)
         (
            ParameterName_as8    := 'Output Value 9',
            ParameterType_u8     := 0,
            attr1_u              := 0,
            attr2_u              := 10000,
            attr3_u              := 50,
            UnitCode_au8         := 15,
            Multiplier_s16       := 1,
            Divisor_s16          := 1,
            NumberOfDigits_u16   := 0,
            AccesslevelCode_u8   := 129,
            attr4_u              := 0,
            EEPROMAddress_s      := (Page_u8 := 3, IntIndex_u8 := 136)
         ),

         (*********************************************)
         (* parameter 3.2.2 *)
         (*********************************************)
         (
            ParameterName_as8    := 'Output Value 10',
            ParameterType_u8     := 0,
            attr1_u              := 0,
            attr2_u              := 10000,
            attr3_u              := 50,
            UnitCode_au8         := 15,
            Multiplier_s16       := 1,
            Divisor_s16          := 1,
            NumberOfDigits_u16   := 0,
            AccesslevelCode_u8   := 129,
            attr4_u              := 0,
            EEPROMAddress_s      := (Page_u8 := 3, IntIndex_u8 := 137)
         ),

         (*********************************************)
         (* parameter 3.2.3 *)
         (*********************************************)
         (
            ParameterName_as8    := 'Output Value 11',
            ParameterType_u8     := 0,
            attr1_u              := 0,
            attr2_u              := 10000,
            attr3_u              := 50,
            UnitCode_au8         := 15,
            Multiplier_s16       := 1,
            Divisor_s16          := 1,
            NumberOfDigits_u16   := 0,
            AccesslevelCode_u8   := 129,
            attr4_u              := 0,
            EEPROMAddress_s      := (Page_u8 := 3, IntIndex_u8 := 138)
         ),

         (*********************************************)
         (* parameter 3.2.4 *)
         (*********************************************)
         (
            ParameterName_as8    := 'Output Value 12',
            ParameterType_u8     := 0,
            attr1_u              := 0,
            attr2_u              := 10000,
            attr3_u              := 50,
            UnitCode_au8         := 15,
            Multiplier_s16       := 1,
            Divisor_s16          := 1,
            NumberOfDigits_u16   := 0,
            AccesslevelCode_u8   := 129,
            attr4_u              := 0,
            EEPROMAddress_s      := (Page_u8 := 3, IntIndex_u8 := 139)
         ),

         (*********************************************)
         (* parameter 3.2.5 *)
         (*********************************************)
         (
            ParameterName_as8    := 'Output Value 13',
            ParameterType_u8     := 0,
            attr1_u              := 0,
            attr2_u              := 10000,
            attr3_u              := 50,
            UnitCode_au8         := 15,
            Multiplier_s16       := 1,
            Divisor_s16          := 1,
            NumberOfDigits_u16   := 0,
            AccesslevelCode_u8   := 129,
            attr4_u              := 0,
            EEPROMAddress_s      := (Page_u8 := 3, IntIndex_u8 := 140)
         ),

         (*********************************************)
         (* parameter 3.2.6 *)
         (*********************************************)
         (
            ParameterName_as8    := 'Output Value 14',
            ParameterType_u8     := 0,
            attr1_u              := 0,
            attr2_u              := 10000,
            attr3_u              := 50,
            UnitCode_au8         := 15,
            Multiplier_s16       := 1,
            Divisor_s16          := 1,
            NumberOfDigits_u16   := 0,
            AccesslevelCode_u8   := 129,
            attr4_u              := 0,
            EEPROMAddress_s      := (Page_u8 := 3, IntIndex_u8 := 141)
         ),

         (*********************************************)
         (* parameter 3.2.7 *)
         (*********************************************)
         (
            ParameterName_as8    := 'Output Value 15',
            ParameterType_u8     := 0,
            attr1_u              := 0,
            attr2_u              := 10000,
            attr3_u              := 50,
            UnitCode_au8         := 15,
            Multiplier_s16       := 1,
            Divisor_s16          := 1,
            NumberOfDigits_u16   := 0,
            AccesslevelCode_u8   := 129,
            attr4_u              := 0,
            EEPROMAddress_s      := (Page_u8 := 3, IntIndex_u8 := 142)
         ),

         (*********************************************)
         (* parameter 3.2.8 *)
         (*********************************************)
         (
            ParameterName_as8    := 'Output Value 16',
            ParameterType_u8     := 0,
            attr1_u              := 0,
            attr2_u              := 10000,
            attr3_u              := 50,
            UnitCode_au8         := 15,
            Multiplier_s16       := 1,
            Divisor_s16          := 1,
            NumberOfDigits_u16   := 0,
            AccesslevelCode_u8   := 129,
            attr4_u              := 0,
            EEPROMAddress_s      := (Page_u8 := 3, IntIndex_u8 := 143)
         )

      ),

      (*********************************************)
      (* parameter group 3.3 - up to 8 parameters can be defined here *)
      (*********************************************)
      (
         GroupName_as8   := 'Output Value 17-36',

         Param_as        := 

         (*********************************************)
         (* parameter 3.3.1 *)
         (*********************************************)
         (
            ParameterName_as8    := 'Output Value 17',
            ParameterType_u8     := 0,
            attr1_u              := 0,
            attr2_u              := 10000,
            attr3_u              := 50,
            UnitCode_au8         := 15,
            Multiplier_s16       := 1,
            Divisor_s16          := 1,
            NumberOfDigits_u16   := 0,
            AccesslevelCode_u8   := 129,
            attr4_u              := 0,
            EEPROMAddress_s      := (Page_u8 := 3, IntIndex_u8 := 144)
         ),

         (*********************************************)
         (* parameter 3.3.2 *)
         (*********************************************)
         (
            ParameterName_as8    := 'Output Value 18',
            ParameterType_u8     := 0,
            attr1_u              := 0,
            attr2_u              := 10000,
            attr3_u              := 50,
            UnitCode_au8         := 15,
            Multiplier_s16       := 1,
            Divisor_s16          := 1,
            NumberOfDigits_u16   := 0,
            AccesslevelCode_u8   := 129,
            attr4_u              := 0,
            EEPROMAddress_s      := (Page_u8 := 3, IntIndex_u8 := 145)
         ),

         (*********************************************)
         (* parameter 3.3.3 *)
         (*********************************************)
         (
         ),

         (*********************************************)
         (* parameter 3.3.4 *)
         (*********************************************)
         (
         ),

         (*********************************************)
         (* parameter 3.3.5 *)
         (*********************************************)
         (
            ParameterName_as8    := 'Output Value 33',
            ParameterType_u8     := 0,
            attr1_u              := 0,
            attr2_u              := 10000,
            attr3_u              := 50,
            UnitCode_au8         := 15,
            Multiplier_s16       := 1,
            Divisor_s16          := 1,
            NumberOfDigits_u16   := 0,
            AccesslevelCode_u8   := 129,
            attr4_u              := 0,
            EEPROMAddress_s      := (Page_u8 := 3, IntIndex_u8 := 148)
         ),

         (*********************************************)
         (* parameter 3.3.6 *)
         (*********************************************)
         (
            ParameterName_as8    := 'Output Value 34',
            ParameterType_u8     := 0,
            attr1_u              := 0,
            attr2_u              := 10000,
            attr3_u              := 50,
            UnitCode_au8         := 15,
            Multiplier_s16       := 1,
            Divisor_s16          := 1,
            NumberOfDigits_u16   := 0,
            AccesslevelCode_u8   := 129,
            attr4_u              := 0,
            EEPROMAddress_s      := (Page_u8 := 3, IntIndex_u8 := 149)
         ),

         (*********************************************)
         (* parameter 3.3.7 *)
         (*********************************************)
         (
            ParameterName_as8    := 'Output Value 35',
            ParameterType_u8     := 0,
            attr1_u              := 0,
            attr2_u              := 10000,
            attr3_u              := 50,
            UnitCode_au8         := 15,
            Multiplier_s16       := 1,
            Divisor_s16          := 1,
            NumberOfDigits_u16   := 0,
            AccesslevelCode_u8   := 129,
            attr4_u              := 0,
            EEPROMAddress_s      := (Page_u8 := 3, IntIndex_u8 := 150)
         ),

         (*********************************************)
         (* parameter 3.3.8 *)
         (*********************************************)
         (
            ParameterName_as8    := 'Output Value 36',
            ParameterType_u8     := 0,
            attr1_u              := 0,
            attr2_u              := 10000,
            attr3_u              := 50,
            UnitCode_au8         := 15,
            Multiplier_s16       := 1,
            Divisor_s16          := 1,
            NumberOfDigits_u16   := 0,
            AccesslevelCode_u8   := 129,
            attr4_u              := 0,
            EEPROMAddress_s      := (Page_u8 := 3, IntIndex_u8 := 151)
         )

      ),

      (*********************************************)
      (* parameter group 3.4 - up to 8 parameters can be defined here *)
      (*********************************************)
      (
         GroupName_as8   := 'Output Value 37-44',

         Param_as        := 

         (*********************************************)
         (* parameter 3.4.1 *)
         (*********************************************)
         (
            ParameterName_as8    := 'Output Value 37',
            ParameterType_u8     := 0,
            attr1_u              := 0,
            attr2_u              := 10000,
            attr3_u              := 50,
            UnitCode_au8         := 15,
            Multiplier_s16       := 1,
            Divisor_s16          := 1,
            NumberOfDigits_u16   := 0,
            AccesslevelCode_u8   := 129,
            attr4_u              := 0,
            EEPROMAddress_s      := (Page_u8 := 3, IntIndex_u8 := 152)
         ),

         (*********************************************)
         (* parameter 3.4.2 *)
         (*********************************************)
         (
            ParameterName_as8    := 'Output Value 38',
            ParameterType_u8     := 0,
            attr1_u              := 0,
            attr2_u              := 10000,
            attr3_u              := 50,
            UnitCode_au8         := 15,
            Multiplier_s16       := 1,
            Divisor_s16          := 1,
            NumberOfDigits_u16   := 0,
            AccesslevelCode_u8   := 129,
            attr4_u              := 0,
            EEPROMAddress_s      := (Page_u8 := 3, IntIndex_u8 := 153)
         ),

         (*********************************************)
         (* parameter 3.4.3 *)
         (*********************************************)
         (
            ParameterName_as8    := 'Output Value 39',
            ParameterType_u8     := 0,
            attr1_u              := 0,
            attr2_u              := 10000,
            attr3_u              := 50,
            UnitCode_au8         := 15,
            Multiplier_s16       := 1,
            Divisor_s16          := 1,
            NumberOfDigits_u16   := 0,
            AccesslevelCode_u8   := 129,
            attr4_u              := 0,
            EEPROMAddress_s      := (Page_u8 := 3, IntIndex_u8 := 154)
         ),

         (*********************************************)
         (* parameter 3.4.4 *)
         (*********************************************)
         (
            ParameterName_as8    := 'Output Value 40',
            ParameterType_u8     := 0,
            attr1_u              := 0,
            attr2_u              := 10000,
            attr3_u              := 50,
            UnitCode_au8         := 15,
            Multiplier_s16       := 1,
            Divisor_s16          := 1,
            NumberOfDigits_u16   := 0,
            AccesslevelCode_u8   := 129,
            attr4_u              := 0,
            EEPROMAddress_s      := (Page_u8 := 3, IntIndex_u8 := 155)
         ),

         (*********************************************)
         (* parameter 3.4.5 *)
         (*********************************************)
         (
            ParameterName_as8    := 'Output Value 41',
            ParameterType_u8     := 0,
            attr1_u              := 0,
            attr2_u              := 10000,
            attr3_u              := 50,
            UnitCode_au8         := 15,
            Multiplier_s16       := 1,
            Divisor_s16          := 1,
            NumberOfDigits_u16   := 0,
            AccesslevelCode_u8   := 129,
            attr4_u              := 0,
            EEPROMAddress_s      := (Page_u8 := 3, IntIndex_u8 := 156)
         ),

         (*********************************************)
         (* parameter 3.4.6 *)
         (*********************************************)
         (
            ParameterName_as8    := 'Output Value 42',
            ParameterType_u8     := 0,
            attr1_u              := 0,
            attr2_u              := 10000,
            attr3_u              := 50,
            UnitCode_au8         := 15,
            Multiplier_s16       := 1,
            Divisor_s16          := 1,
            NumberOfDigits_u16   := 0,
            AccesslevelCode_u8   := 129,
            attr4_u              := 0,
            EEPROMAddress_s      := (Page_u8 := 3, IntIndex_u8 := 157)
         ),

